# EPICS substitutions: ek9000App/Db/EL3154.substitutions
file EL3154.template
{       pattern
        {
                TERMINAL,

        }
        {
        }
}
